{attribute 'GeneratedUsingTerminal: ATH2000-0250-0023'}
{attribute addProperty BoxType "ATH2000-0250-0023"}
{attribute addProperty Id "A_0015_ATH2040_5250_0022ATH2040_41437DDC14"}
{attribute addProperty CRC "3861582314"}
{attribute addProperty Size "14"}
TYPE A_0002_ATH2000_0250_0023_E62B11EA EXTENDS ATH2000_2EA6C9BF :
STRUCT
	{attribute addProperty Name "A_0015_ATH2040_5250_0022"}
	{attribute addProperty PreviousPort "A_0002(ATH2000-0250-0023) : B"}
	A_0015_ATH2040_5250_0022 : ATH2040_41437DDC;
END_STRUCT
END_TYPE

(* stored: Version 1.2.0.0, ProductVersion 3.1.4024.9
   DUT A_0002_ATH2000_0250_0023_E62B11EA: Id {531a2732-6bc3-4037-9ec2-6f9cda82e4fd} *)
